Fanuc KAREL source: SELECT_TPE.kl

PROGRAM T
%NOLOCKGROUP
VAR
 v0 : STRING[40]
 v1 : INTEGER
BEGIN
 SELECT_TPE(v0, v1)
END T
